# EPICS autosave request: oxfordApp/Db/oxford_settings.req
$(P)KVP
$(P)KVP_MAX
$(P)KVP_MIN
$(P)WATT
$(P)WATT_MAX
$(P)WATT_MIN
$(P)PULSE_WIDTH
$(P)AUTOKILL_LENGTH
